% RSLogix 500 project Logic Gates.RSS, saved by version 8.30.00.16 %
PROJECT "UNTITLED"    % processor: Bul.1763 MicroLogix 1100 Series B %

PROGRAM FILES
  LAD 2   6 rungs

DATA FILES
  O0 OUTPUT  4 elements
  I1 INPUT  6 elements
  S2 STATUS  66 elements
  B3 BINARY  1 elements
  T4 TIMER  1 elements
  C5 COUNTER  1 elements
  R6 CONTROL  1 elements
  N7 INTEGER  1 elements
  F8 FLOAT  1 elements

LADDER 2
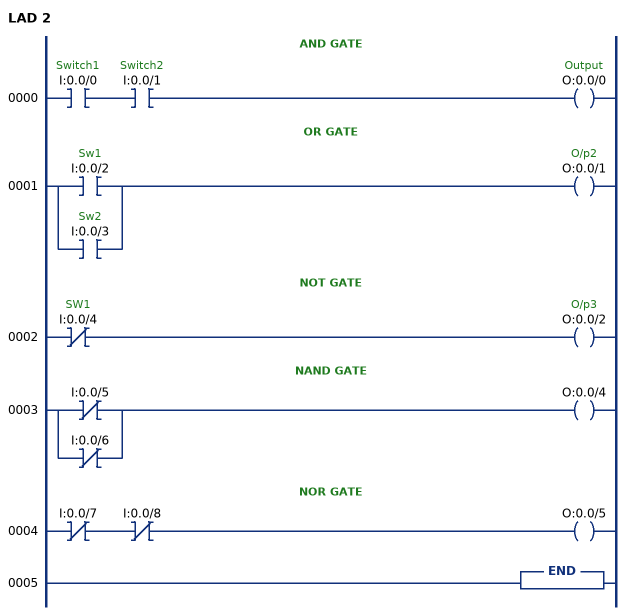
% Rung: 0 %
% TITLE: AND GATE %
SOR XIC I:0.0/0 XIC I:0.0/1 OTE O:0.0/0 EOR
%   I:0.0/0  "Switch1" %
%   I:0.0/1  "Switch2" %
%   O:0.0/0  "Output" %
% Rung: 1 %
% TITLE: OR GATE %
SOR BST XIC I:0.0/2 NXB XIC I:0.0/3 BND OTE O:0.0/1 EOR
%   I:0.0/2  "Sw1" %
%   I:0.0/3  "Sw2" %
%   O:0.0/1  "O/p2" %
% Rung: 2 %
% TITLE: NOT GATE %
SOR XIO I:0.0/4 OTE O:0.0/2 EOR
%   I:0.0/4  "SW1" %
%   O:0.0/2  "O/p3" %
% Rung: 3 %
% TITLE: NAND GATE %
SOR BST XIO I:0.0/5 NXB XIO I:0.0/6 BND OTE O:0.0/4 EOR
% Rung: 4 %
% TITLE: NOR GATE %
SOR XIO I:0.0/7 XIO I:0.0/8 OTE O:0.0/5 EOR
% Rung: 5 %
SOR END EOR

OTHER DOCUMENTED ADDRESSES
  I:1.0/0  "Switch1"
  I:1.0/1  "Switch2"
  O:1.0/0  "Output"
